TYPE ST_JointBenchAds :
STRUCT
    bEnable : BOOL;
    bStart : BOOL;
    bStop : BOOL;
    bResetFault : BOOL;
    fTargetPositionDeg : LREAL;
    nCommandSequence : DINT;

    bReady : BOOL;
    bBusy : BOOL;
    bDone : BOOL;
    bError : BOOL;
    bOperationEnabled : BOOL;
    bWatchdogOk : BOOL;

    fActualPositionDeg : LREAL;
    fActualVelocityDps : LREAL;
    fFollowingErrorDeg : LREAL;
    fCurrentA : LREAL;
    fTemperatureC : LREAL;

    nStatusword : DINT;
    nControlword : DINT;
    nFaultCode : DINT;
    nErrorCode : DINT;

    sDeviceName : STRING(80);
    nVendorId : DINT;
    nProductCode : DINT;
    nRevision : DINT;
END_STRUCT
END_TYPE

TYPE ST_Ti5CiA402PdoInput :
STRUCT
    nStatusword : UINT;
    nActualPosition : DINT;
    nActualVelocity : DINT;
    nActualTorqueOrCurrent : INT;
    nErrorCode : UINT;
    nTemperatureRaw : INT;
END_STRUCT
END_TYPE

TYPE ST_Ti5CiA402PdoOutput :
STRUCT
    nControlword : UINT;
    nModeOfOperation : SINT;
    nTargetPosition : DINT;
END_STRUCT
END_TYPE

(* stored: Version 1.1.0.1, ProductVersion 3.1.4024.0 *)
